FUNCTION_BLOCK SET_SPINDLE_DATA (* Sets spindle speed data to machine *)
  (* Standard: 61499-2 *)
  (* Version 1.0, 18-04-2012, GASR, Universidade do Estado de Santa Catarina *)
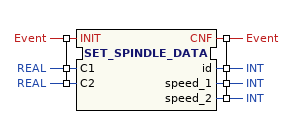
  EVENT_INPUT
    INIT WITH C1, C2;
  END_EVENT
  EVENT_OUTPUT
    CNF WITH id, speed_1, speed_2;
  END_EVENT
  VAR_INPUT
    C1 : REAL; (* Coeficient 1 *)
    C2 : REAL; (* Coeficient 2 *)
  END_VAR
  VAR_OUTPUT
    id : INT;
    speed_1 : INT;
    speed_2 : INT;
  END_VAR
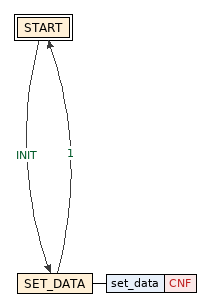
  EC_STATES
    START;
    SET_DATA : set_data -> CNF;
  END_STATES
  EC_TRANSITIONS
    START TO SET_DATA := INIT;
    SET_DATA TO START := 1;
  END_TRANSITIONS
  ALGORITHM set_data IN Lua:
id = C1
local precision = 3
speed_1 = math.floor( C2 )
speed_2 = (C2 - speed_1)*(10^precision)
speed_2 = math.floor( speed_2 )
  END_ALGORITHM
END_FUNCTION_BLOCK
